ABB RAPID module: JSD.mod

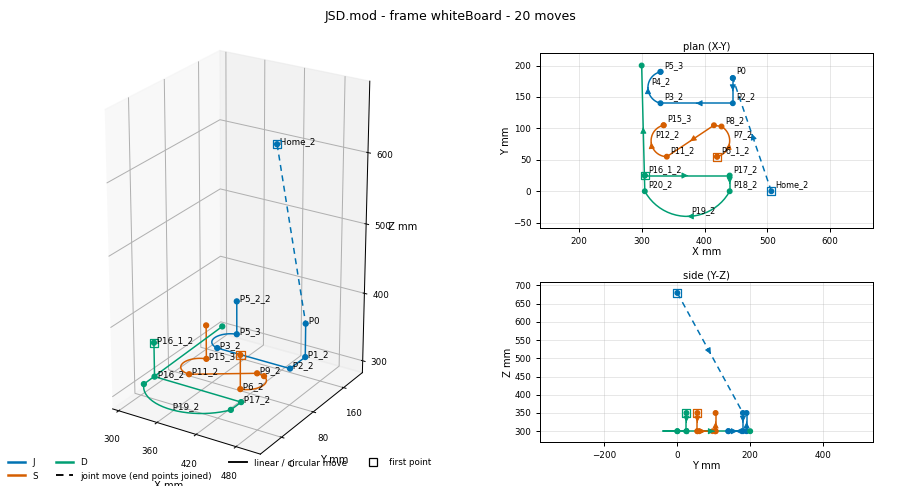
[picture p0: tool path of JSD.mod in frame whiteBoard, 20 of 20 moves have a stored position in this frame; points joined in program order, loops and branches not executed]
MODULE JSD
     CONST robtarget Home:=[[506.291651246,0,679.5],[0.5,0,0.866025404,0],[0,0,0,0],[9E+09,9E+09,9E+09,9E+09,9E+09,9E+09]];

        !J points
        CONST robtarget UCS:=[[350,200,300],[0,0,1,0],[0,0,0,0],[9E+09,9E+09,9E+09,9E+09,9E+09,9E+09]];
        CONST robtarget P1:=[[640,160,300],[0,0,1,0],[0,0,0,0],[9E+09,9E+09,9E+09,9E+09,9E+09,9E+09]];
        CONST robtarget P2:=[[640,80,300],[0,0,1,0],[0,0,0,0],[9E+09,9E+09,9E+09,9E+09,9E+09,9E+09]];
        CONST robtarget P3:=[[410,80,300],[0,0,1,0],[0,0,0,0],[9E+09,9E+09,9E+09,9E+09,9E+09,9E+09]];
        CONST robtarget P4:=[[370,130,300],[0,0,1,0],[0,0,0,0],[9E+09,9E+09,9E+09,9E+09,9E+09,9E+09]];
        CONST robtarget P5:=[[410,180,300],[0,0,1,0],[0,0,0,0],[9E+09,9E+09,9E+09,9E+09,9E+09,9E+09]];
        CONST robtarget P5_2:=[[410,180,350],[0,0,1,0],[0,0,0,0],[9E+09,9E+09,9E+09,9E+09,9E+09,9E+09]];

        !S points
        CONST robtarget P6_1:=[[590,-90,350],[0,0,1,0],[0,0,0,0],[9E+09,9E+09,9E+09,9E+09,9E+09,9E+09]];
        CONST robtarget P6:=[[540,-90,300],[0,0,1,0],[-1,0,-1,0],[9E+09,9E+09,9E+09,9E+09,9E+09,9E+09]];
        CONST robtarget P7:=[[630,-40,300],[0,0,1,0],[-1,0,-1,0],[9E+09,9E+09,9E+09,9E+09,9E+09,9E+09]];
        CONST robtarget P8:=[[604,6,300],[0,0,1,0],[0,0,0,0],[9E+09,9E+09,9E+09,9E+09,9E+09,9E+09]];
        CONST robtarget P9:=[[580,10,300],[0,0,1,0],[0,0,0,0],[9E+09,9E+09,9E+09,9E+09,9E+09,9E+09]];
        CONST robtarget P11:=[[430,-90,300],[0,0,1,0],[-1,0,-1,0],[9E+09,9E+09,9E+09,9E+09,9E+09,9E+09]];
        CONST robtarget P12:=[[400,-90,300],[0,0,1,0],[-1,0,-1,0],[9E+09,9E+09,9E+09,9E+09,9E+09,9E+09]];
        CONST robtarget P13:=[[360,-40,300],[0,0,1,0],[1,2,-1,6],[9E+09,9E+09,9E+09,9E+09,9E+09,9E+09]];
        CONST robtarget P14:=[[375,-10,300],[0,0,1,0],[1,2,-1,6],[9E+09,9E+09,9E+09,9E+09,9E+09,9E+09]];
        CONST robtarget P15:=[[420,10,300],[0,0,1,0],[0,0,0,0],[9E+09,9E+09,9E+09,9E+09,9E+09,9E+09]];
        CONST robtarget P15_2:=[[420,10,350],[0,0,1,0],[0,0,0,0],[9E+09,9E+09,9E+09,9E+09,9E+09,9E+09]];
        CONST robtarget P16_1:=[[360,-150,350],[0,0,1,0],[0,0,0,0],[9E+09,9E+09,9E+09,9E+09,9E+09,9E+09]];
        CONST robtarget P16:=[[360,-150,300],[0,0,1,0],[-1,0,-1,0],[9E+09,9E+09,9E+09,9E+09,9E+09,9E+09]];
        CONST robtarget P17:=[[630,-150,300],[0,0,1,0],[-1,0,-1,0],[9E+09,9E+09,9E+09,9E+09,9E+09,9E+09]];
        CONST robtarget P18:=[[630,-200,300],[0,0,1,0],[-1,0,-1,0],[9E+09,9E+09,9E+09,9E+09,9E+09,9E+09]];
        CONST robtarget P19:=[[496,-280,300],[0,0,1,0],[-1,0,-1,0],[9E+09,9E+09,9E+09,9E+09,9E+09,9E+09]];
        CONST robtarget P20:=[[360,-200,300],[0,0,1,0],[-1,0,-1,0],[9E+09,9E+09,9E+09,9E+09,9E+09,9E+09]];
        CONST robtarget Home_2:=[[506.291651246,0,679.5],[0.5,0,0.866025404,0],[0,0,0,0],[9E+09,9E+09,9E+09,9E+09,9E+09,9E+09]];
        CONST robtarget P5_2_2:=[[330,190,350],[0,0,1,0],[0,0,0,0],[9E+09,9E+09,9E+09,9E+09,9E+09,9E+09]];
        CONST robtarget P5_3:=[[330,190,300],[0,0,1,0],[0,0,0,0],[9E+09,9E+09,9E+09,9E+09,9E+09,9E+09]];
        CONST robtarget P2_2:=[[445,140,300],[0,0,1,0],[0,0,0,0],[9E+09,9E+09,9E+09,9E+09,9E+09,9E+09]];
        CONST robtarget P3_2:=[[330,140,300],[0,0,1,0],[0,0,0,0],[9E+09,9E+09,9E+09,9E+09,9E+09,9E+09]];
        CONST robtarget P4_2:=[[310,165,300],[0,0,1,0],[0,0,0,0],[9E+09,9E+09,9E+09,9E+09,9E+09,9E+09]];
        CONST robtarget P1_2:=[[445,180,300],[0,0,1,0],[0,0,0,0],[9E+09,9E+09,9E+09,9E+09,9E+09,9E+09]];
        CONST robtarget P0:=[[445,180,350],[0,0,1,0],[0,0,0,0],[9E+09,9E+09,9E+09,9E+09,9E+09,9E+09]];
        CONST robtarget P6_1_2:=[[420,55,350],[0,0,1,0],[0,0,0,0],[9E+09,9E+09,9E+09,9E+09,9E+09,9E+09]];
        CONST robtarget P6_2:=[[420,55,300],[0,0,1,0],[0,0,0,0],[9E+09,9E+09,9E+09,9E+09,9E+09,9E+09]];
        CONST robtarget P15_3:=[[335,105,300],[0,0,1,0],[0,0,0,0],[9E+09,9E+09,9E+09,9E+09,9E+09,9E+09]];
        CONST robtarget P8_2:=[[427,103,300],[0,0,1,0],[0,0,0,0],[9E+09,9E+09,9E+09,9E+09,9E+09,9E+09]];
        CONST robtarget P7_2:=[[440,80,300],[0,0,1,0],[0,0,0,0],[9E+09,9E+09,9E+09,9E+09,9E+09,9E+09]];
        CONST robtarget P9_2:=[[415,105,300],[0,0,1,0],[0,0,0,0],[9E+09,9E+09,9E+09,9E+09,9E+09,9E+09]];
        CONST robtarget P15_2_2:=[[335,105,350],[0,0,1,0],[0,0,0,0],[9E+09,9E+09,9E+09,9E+09,9E+09,9E+09]];

        !D points
        CONST robtarget P13_2:=[[305,80,300],[0,0,1,0],[-2,-2,0,6],[9E+09,9E+09,9E+09,9E+09,9E+09,9E+09]];
        CONST robtarget P14_2:=[[425,95,300],[0,0,1,0],[-2,-2,0,6],[9E+09,9E+09,9E+09,9E+09,9E+09,9E+09]];
        CONST robtarget P12_2:=[[315,80,300],[0,0,1,0],[0,0,0,0],[9E+09,9E+09,9E+09,9E+09,9E+09,9E+09]];
        CONST robtarget P11_2:=[[340,55,300],[0,0,1,0],[0,0,0,0],[9E+09,9E+09,9E+09,9E+09,9E+09,9E+09]];
        CONST robtarget UCS_2:=[[300,200,300],[0,0,1,0],[0,0,0,0],[9E+09,9E+09,9E+09,9E+09,9E+09,9E+09]];
        CONST robtarget P16_1_2:=[[305,25,350],[0,0,1,0],[0,0,0,0],[9E+09,9E+09,9E+09,9E+09,9E+09,9E+09]];
        CONST robtarget P16_2:=[[305,25,300],[0,0,1,0],[0,0,0,0],[9E+09,9E+09,9E+09,9E+09,9E+09,9E+09]];
        CONST robtarget P17_2:=[[440,25,300],[0,0,1,0],[0,0,0,0],[9E+09,9E+09,9E+09,9E+09,9E+09,9E+09]];
        CONST robtarget P18_2:=[[440,0,300],[0,0,1,0],[0,0,0,0],[9E+09,9E+09,9E+09,9E+09,9E+09,9E+09]];
        CONST robtarget P19_2:=[[373,-40,300],[0,0,1,0],[0,0,0,0],[9E+09,9E+09,9E+09,9E+09,9E+09,9E+09]];
        CONST robtarget P20_2:=[[305,0,300],[0,0,1,0],[0,0,0,0],[9E+09,9E+09,9E+09,9E+09,9E+09,9E+09]];



        PROC J()
            MoveJ Home_2,v500,z100,tool0\WObj:=whiteBoard;
            MoveJ P0,v500,z100,tool0\WObj:=whiteBoard;
            MoveL P1_2,v100,z100,tool0\WObj:=whiteBoard;
            MoveL P2_2,v100,z0,tool0\WObj:=whiteBoard;
            MoveL P3_2,v100,z0,tool0\WObj:=whiteBoard;
            MoveC P4_2,P5_3,v100,z0,tool0\WObj:=whiteBoard;
            MoveL P5_2_2,v100,z0,tool0\WObj:=whiteBoard;
        ENDPROC
        !PROC main()
        !ENDPROC
        PROC S()
            MoveJ P6_1_2,v500,z0,tool0\WObj:=whiteBoard;
            MoveL P6_2,v100,z0,tool0\WObj:=whiteBoard;
            MoveC P7_2,P8_2,v100,z0,tool0\WObj:=whiteBoard;
            MoveL P9_2,v100,z0,tool0\WObj:=whiteBoard;
            MoveL P11_2,v100,z0,tool0\WObj:=whiteBoard;
            MoveC P12_2,P15_3,v100,z0,tool0\WObj:=whiteBoard;

            MoveL P15_2_2,v100,z0,tool0\WObj:=whiteBoard;
        ENDPROC
        PROC D()
            MoveJ P16_1_2,v500,z0,tool0\WObj:=whiteBoard;
            MoveL P16_2,v100,z0,tool0\WObj:=whiteBoard;
            MoveL P17_2,v100,z0,tool0\WObj:=whiteBoard;
            MoveL P18_2,v100,z0,tool0\WObj:=whiteBoard;
            MoveC P19_2,P20_2,v100,z0,tool0\WObj:=whiteBoard;
            MoveL UCS_2,v100,z0,tool0\WObj:=whiteBoard;
        ENDPROC
        PROC pathJSD()
            J;
            S;
            D;
        ENDPROC
    ENDMODULE
